// Mitsubishi GX Works2 project: 传数值的另一种写法   PLC: L02S

FUNCTION_BLOCK xsz
VAR_INPUT
  IN1 : BOOL;
END_VAR
VAR_OUTPUT
  OUT1 : BOOL;
END_VAR
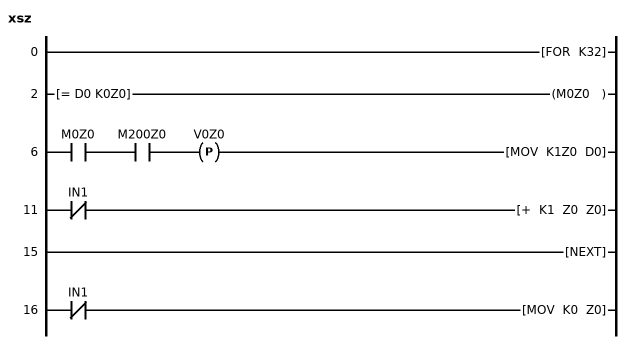
0     FOR     K32
2     LD=     D0 K0Z0
      OUT     M0Z0
6     LD      M0Z0
      AND     M200Z0
      EGP     V0Z0
      MOV     K1Z0 D0
11    LDI     IN1
      +       K1 Z0 Z0
15    NEXT
16    LDI     IN1
      MOV     K0 Z0
END_FUNCTION_BLOCK

PROGRAM xszxsz
VAR
  xsz_1 : xsz;
END_VAR
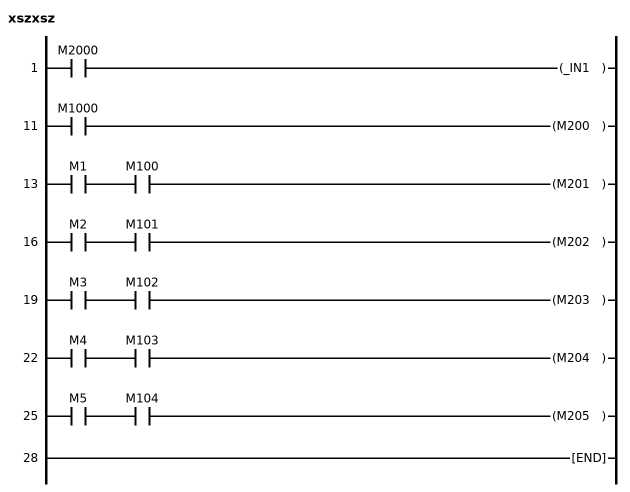
; FB BLK START xsz(xsz_1)
1     LD      M2000
      OUT     _IN1
; FB START
; FB_NAME xsz
; INSTANCE_NAME xsz_1
; FB IN_B:IN1
; FB OUT_OUT1:B
; FB END
; FB BLK END
11    LD      M1000
      OUT     M200
13    LD      M1
      AND     M100
      OUT     M201
16    LD      M2
      AND     M101
      OUT     M202
19    LD      M3
      AND     M102
      OUT     M203
22    LD      M4
      AND     M103
      OUT     M204
25    LD      M5
      AND     M104
      OUT     M205
28    END
END_PROGRAM
